ABB RAPID module: YuMiLib_Params_R.sys

MODULE YuMiLib_Params_R(SYSMODULE)

    !***************************************************************************
    !*                              Common parameters                          *
    !***************************************************************************
    CONST loaddata ld_YuMiGripper_S:=[0.230,[8.2,11.7,52.0],[1,0,0,0],0.00021,0.00024,0.00009];
    CONST loaddata ld_YuMiGripper_S_V1:=[0.248,[8.6,11.7,52.7],[1,0,0,0],0.00021,0.00024,0.00009];
    CONST loaddata ld_YuMiGripper_S_V1_V2:=[0.280,[7.1,11.9,47.3],[1,0,0,0],0.00025,0.00029,0.00012];
    CONST loaddata ld_YuMiGripper_S_C:=[0.244,[7.5,11.8,52.7],[1,0,0,0],0.00021,0.00023,0.00008];
    CONST loaddata ld_YuMiGripper_S_C_V1:=[0.262,[7.8,11.9,50.7],[1,0,0,0],0.00022,0.00024,0.00009];

    !**********************************
    !**********Standard parameters needed for Camera Calibration **********************************************
    !***Do not change these.
    CONST string markerFinderJob:="PatternABB.job";
    TASK PERS num HandCamera_Kinv{3,3}:=[[0.000584319,2.15201E-06,-0.388731],[0,0.000582727,-0.29143],[0,0,1]];
    TASK PERS num HandCamera_K{3,3}:=[[1711.39,-6.32017,663.43],[0,1716.07,500.114],[0,0,1]];
    TASK PERS tooldata tHandCamera:=[TRUE,[[-7.22594,27.6025,35.0158],[0.507289,-0.493481,-0.498638,-0.500495]],[0.262,[7.8,11.9,50.7],[1,0,0,0],0.00022,0.00024,9E-05]];
    CONST pose peDefault_tFrame_HandCamera:=[[-7.3, 28.3, 35.1], [0.5, -0.5, -0.5, -0.5]];
    CONST pose peDefault_tFrame_ABBLogo:=[[0, -28.3, 30], [0.5, -0.5, -0.5, -0.5]];
    TASK PERS wobjdata WObj_Vision:=[FALSE,TRUE,"",[[401.591,32.4092,0],[0.424655,-1.21554E-07,-1.90773E-07,0.905355]],[[0,0,0],[1,0,0,0]]];

    ! Predefined tools for different configurations of the Standard Smart Gripper
	TASK PERS tooldata tGripper:=[TRUE,[[-0.214928,0.306602,135.552],[1,0,0,0]],[0.23,[8.2,11.7,52],[1,0,0,0],0.00021,0.00024,9E-05]];
	TASK PERS tooldata tVacuum1:=[TRUE,[[63.5,18.5,37.5],[0.707106781,0,0.707106781,0]],[0.248,[8.6,11.7,52.7],[1,0,0,0],0.00021,0.00024,0.00009]];
	TASK PERS tooldata tVacuum2:=[TRUE,[[-63.5,18.5,37.5],[0.707106781,0,-0.707106781,0]],[0.280,[7.1,11.9,47.3],[1,0,0,0],0.00025,0.00029,0.00012]];

    !***************************************************************************
    !*                         Task specific paramters                         *
    !***************************************************************************

    TASK PERS string YuMiLib_CameraName:="HandCameraR";

    CONST robtarget pCamera_Calib_Near:=[[413,-50,400],[1,0,0,0],[1,0,2,4],[-110,9E+09,9E+09,9E+09,9E+09,9E+09]];
    CONST robtarget pCamera_Calib_Far:=[[413,-250,400],[1,0,0,0],[1,0,2,4],[-110,9E+09,9E+09,9E+09,9E+09,9E+09]];
    CONST robtarget pCamera_Calib_train:=[[400,-175,380],[1,0,0,0],[1,0,1,4],[-110,9E+09,9E+09,9E+09,9E+09,9E+09]];

    CONST robtarget pShowABBLogo:=[[405+15,-150,405],[0,0,0,1],[1,0,-1,4],[-110,9E+09,9E+09,9E+09,9E+09,9E+09]];

    TASK PERS wobjdata WObj_FollowRobL:=[FALSE,FALSE,"ROB_L",[[0, 0, 0],[1, 0, 0, 0]],[[0, 0, 0],[1, 0, 0, 0]]];


    !**************************************************************************
    !*                                Speeddata                               *
    !**************************************************************************
    CONST speeddata vSlow:=[100,50,5000,1000];
    CONST speeddata vMedium:=[300,150,5000,1000];
    CONST speeddata vFast:=v1000;

ENDMODULE
